PROGRAM Axis01_Status
VAR
//Motor
	Axis01_Status: MC_ReadStatus;
	Axis01_Position_Read: MC_ReadActualPosition;
	Axis01_Velocity_Read: MC_ReadActualVelocity;
	Axis01_Reset: MC_Reset;
	Axis01_Stop: MC_Stop;
//System_Bit
	Always_ON	:	BOOL	:=TRUE	;//상시 ON 
	Always_OFF	:	BOOL	:=FALSE	;//상시 OFF

END_VAR

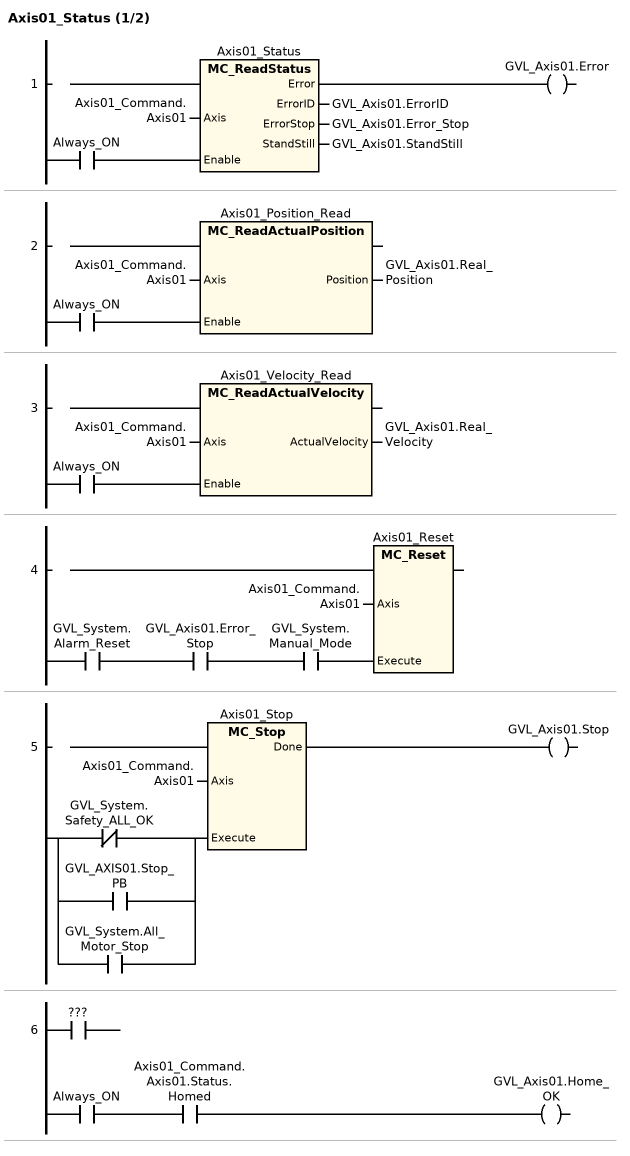
// NETWORK 1
Axis01_Status(
    Axis := Axis01_Command.Axis01,
    Enable := Always_ON,
    Error => GVL_Axis01.Error,
    ErrorID => GVL_Axis01.ErrorID,
    ErrorStop => GVL_Axis01.Error_Stop,
    StandStill => GVL_Axis01.StandStill); // MC_ReadStatus

// NETWORK 2
Axis01_Position_Read(
    Axis := Axis01_Command.Axis01,
    Enable := Always_ON,
    Position => GVL_Axis01.Real_Position); // MC_ReadActualPosition

// NETWORK 3
Axis01_Velocity_Read(
    Axis := Axis01_Command.Axis01,
    Enable := Always_ON,
    ActualVelocity => GVL_Axis01.Real_Velocity); // MC_ReadActualVelocity

// NETWORK 4
Axis01_Reset(Axis := Axis01_Command.Axis01, Execute := GVL_System.Alarm_Reset AND GVL_Axis01.Error_Stop AND GVL_System.Manual_Mode); // MC_Reset

// NETWORK 5
Axis01_Stop(Axis := Axis01_Command.Axis01, Execute := NOT GVL_System.Safety_ALL_OK OR GVL_AXIS01.Stop_PB OR GVL_System.All_Motor_Stop); // MC_Stop
GVL_Axis01.Stop := Axis01_Stop.Done;

// NETWORK 6
GVL_Axis01.Home_OK := Always_ON AND Axis01_Command.Axis01.Status.Homed;

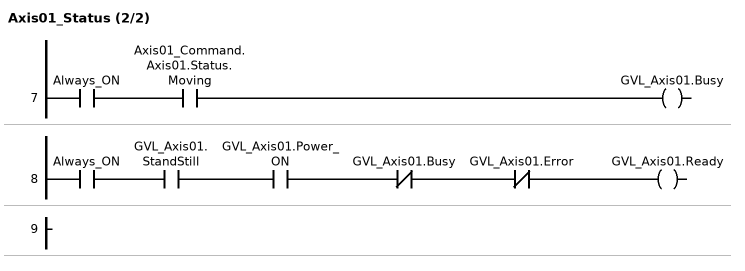
// NETWORK 7
GVL_Axis01.Busy := Always_ON AND Axis01_Command.Axis01.Status.Moving;

// NETWORK 8
GVL_Axis01.Ready := Always_ON AND GVL_Axis01.StandStill AND GVL_Axis01.Power_ON AND NOT GVL_Axis01.Busy AND NOT GVL_Axis01.Error;

// NETWORK 9

END_PROGRAM

(* stored: Version 1.1.0.1, ProductVersion 3.1.4024.15
   POU Axis01_Status: Id {5d0bbb67-15d0-439d-aa4f-15fa70d56d90}, SpecialFunc None *)
